FUNCTION_BLOCK PUBLIC FB_MappingInputs
VAR_INPUT
END_VAR
VAR_OUTPUT
END_VAR
VAR
END_VAR

// Exercice 1
FIO_I_BoutonMarche := FIO_Input1[0];
FIO_I_Capteur := FIO_Input1[1];
FIO_I_BoutonAvancer := FIO_Input1[2];

END_FUNCTION_BLOCK

(* stored: Version 1.1.0.1, ProductVersion 3.1.4024.11
   POU FB_MappingInputs: Id {c1ec172f-2dc8-4773-89ed-4407992e7b38}, SpecialFunc None *)
